(* IEC 61131-3 sources: VeriST/extraction, 6 files *)

(* ---- test_factorial.st ---- *)
(* 阶乘计算程序
   计算 5! = 120
*)
PROGRAM Factorial
VAR
    n : INT := 5;
    result : INT := 1;
    i : INT := 1;
END_VAR

(* 使用循环计算阶乘 *)
WHILE i <= n DO
    result := result * i;
    i := i + 1;
END_WHILE

(* 此时 result = 120 *)
END_PROGRAM

(* ---- test_fibonacci.st ---- *)
(* 斐波那契数列程序
   计算第10个斐波那契数 = 55
*)
PROGRAM Fibonacci
VAR
    n : INT := 10;
    fib_prev : INT := 0;
    fib_curr : INT := 1;
    fib_next : INT;
    counter : INT := 2;
END_VAR

WHILE counter <= n DO
    fib_next := fib_prev + fib_curr;
    fib_prev := fib_curr;
    fib_curr := fib_next;
    counter := counter + 1;
END_WHILE

(* 此时 fib_curr = 55 *)
END_PROGRAM

(* ---- test_gcd.st ---- *)
(* 最大公约数程序
   使用欧几里得算法计算 GCD(48, 18) = 6
*)
PROGRAM GCD
VAR
    a : INT := 48;
    b : INT := 18;
    temp : INT;
END_VAR

WHILE b <> 0 DO
    temp := b;
    b := a MOD b;
    a := temp;
END_WHILE

(* 此时 a = 6 *)
END_PROGRAM

(* ---- test_qint_demo.st ---- *)
PROGRAM test_qint_demo
VAR
    x : QINT;
    y : QINT;
    result : QINT;
END_VAR
    x := 10;
    y := 20;
    result := x + y;
END_PROGRAM

(* ---- test_quality.st ---- *)
PROGRAM test_quality
VAR
    x : QINT;
    y : INT;
    flag : QBOOL;
END_VAR
    y := 100;
    x := 42;
    flag := TRUE;
END_PROGRAM

(* ---- test_simple.st ---- *)
PROGRAM test_simple
VAR
    x : INT;
END_VAR
    x := 42;
END_PROGRAM
